// TIA Portal V15.1 export
// export: Created 2026-01-15T16:29:45.4592346Z, ExportSetting WithDefaults, WithReadOnly, DisplayName Totally Integrated Automation Portal, DisplayVersion V15.1 Update 8, DisplayName TIA Portal Openness, DisplayVersion V15.1 Update 8, DisplayName STEP 7 Professional, DisplayVersion V15.1 Update 8, DisplayName WinCC Advanced, DisplayVersion V15.1 Update 8
FUNCTION_BLOCK "9.TIMER_DELAY"   // FB9, LAD
{ S7_Optimized_Access := 'TRUE' }
VERSION : 0.1
// stored: AutoNumber false, CodeModifiedDate 2025-08-27T17:13:13.1552526Z, CompileDate 2026-01-15T16:25:50.0427227Z, CreationDate 2026-01-15T16:22:49.8270549Z, DownloadWithoutReinit false, HandleErrorsWithinBlock false, InterfaceModifiedDate 2022-05-24T16:36:11.1705081Z, IsConsistent true, IsIECCheckEnabled false, IsKnowHowProtected false, IsRetainMemResEnabled false, IsWriteProtected false, LibraryConformanceStatus The object is library-conformant., MemoryReserve 100, ModifiedDate 2025-08-27T17:13:13.1552526Z, ParameterModified 2022-05-24T16:36:11.1705081Z, PLCSimAdvancedSupport false, SetENOAutomatically False, StructureModified 2022-05-24T16:36:11.1705081Z, UDAEnableTagReadback false
   VAR_INPUT
      ON : Bool;
      CLOCK_1S : Bool;
      T_DELAY : Real;
   END_VAR
   VAR_OUTPUT
      OUT : Bool;
      T_OUT : Real;
   END_VAR
   VAR
      TDL : Real;
      CLK : Bool;
   END_VAR
   VAR_TEMP   // added for the SCL form of the ladder/FBD networks
      _w1 : Bool;
   END_VAR
BEGIN

REGION Network 1
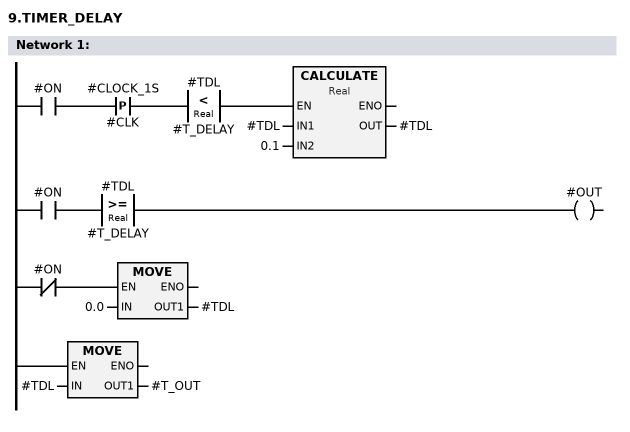
   RUNG wire#powerrail
      Contact( #ON )
      P_Contact(operand := #CLOCK_1S, bit := #CLK)
      { S7_Templates := "SrcType := Real" } LT_Contact(in1 := #TDL, in2 := #T_DELAY)
      { S7_Templates := "SrcType := Real"; S7_Expression := "IN1+IN2" } Calculate(in1 := #TDL, in2 := 0.1, out => #TDL)
   END_RUNG
   RUNG wire#powerrail
      Contact( #ON )
      { S7_Templates := "SrcType := Real" } GE_Contact(in1 := #TDL, in2 := #T_DELAY)
      Coil( #OUT )
   END_RUNG
   RUNG wire#powerrail
      I_Contact( #ON )
      Move(in := 0.0, out1 => #TDL)
   END_RUNG
   RUNG wire#powerrail
      Move(in := #TDL, out1 => #T_OUT)
   END_RUNG
   // the same network as SCL:
   #_w1 := #ON AND #CLOCK_1S AND NOT #CLK;   // rising edge of #CLOCK_1S
   #CLK := #CLOCK_1S;
   IF #_w1 AND (#TDL < #T_DELAY) THEN #TDL := #TDL+0.1; END_IF;
   #OUT := #ON AND (#TDL >= #T_DELAY);
   IF NOT #ON THEN #TDL := 0.0; END_IF;
   #T_OUT := #TDL;
END_REGION
END_FUNCTION_BLOCK
